(* IEC 61131-3 sources: Kur_TemplateProject_v1/TestPanelV1.fbsproj/MyController.device.xml.v3^/Plc Logic.plclogic.xml.v3^/Application.application.xml.v3^/02_GlobalVars, 4 files *)

(* ---- GVL.gvl ---- *)
{attribute 'qualified_only'}
VAR_GLOBAL
END_VAR

(* ---- GVL_IO.gvl ---- *)
VAR_GLOBAL

    // ---------- DIGITAL INPUTS ----------
	(* Buttons *)
    StartButton_In      : BOOL		:= TRUE;
    StopButton_In       : BOOL;
    ResetButton_In      : BOOL		:= TRUE;
    Emergency_In        : BOOL		:= TRUE;     // NC contact -> TRUE = OK

	(* Switchs *)
	ManualMode_Sw		: BOOL;
	AutoMode_Sw			: BOOL		:= TRUE;

    // ---------- DIGITAL OUTPUTS ----------
    (* Lamp *)
	RunLamp_Out       	: BOOL;
	ReadyLamp_Out		: BOOL;
    AlarmLamp_Out       : BOOL;

    // ---------- VIRTUAL MASTER ----------
    MasterAxis  : MOIN.FB_ControlledAxis;

    // ---------- REAL AXES ----------
    MainChain   : MOIN.FB_ControlledAxis;   // DRV1
    Conveyor    : MOIN.FB_ControlledAxis;   // DRV2
    CutterAxis  : MOIN.FB_ControlledAxis;   // DRV3

END_VAR

(* ---- GVL_Recipe.gvl ---- *)
VAR_GLOBAL

	IS_DEBUG: BOOL := TRUE;
END_VAR

(* ---- GVL_System.gvl ---- *)
VAR_GLOBAL

    // ---------- ALARMS ----------
    Alarms      : AlarmSystem;

    // ---------- DATE / TIME ----------
    Clock       : TimeData;
    TimeRead    : BOOL;     // <- HMI button "Load"
    TimeWrite   : BOOL;     // <- HMI button "Apply"

	// --------- SYSTEM --------------
	Machine		: MachineStatus;
END_VAR
